{region '#Template'}
	{attribute 'Version' := '1.2.0.0'}
	{attribute 'Tags' := '"LCID": "1031", "Text": "DUT, Operation mode, Universal, On, Off"'}
	{attribute 'Tags' := '"LCID": "1033", "Text": "DUT, Operation mode, Universal, On, Off"'}
	{attribute 'Description' := '"LCID": "1031", "Text": "Betriebsart Ein Aus"'}
	{attribute 'Description' := '"LCID": "1033", "Text": "Operating on off"'}
{endregion}

{attribute qualified_only}
TYPE E_BA_OnOff :
(
	eOff			:= 1,
	eOn				:= 2
	
) UDINT;
END_TYPE

(* stored: Version 1.1.0.1, ProductVersion 3.1.4024.9
   DUT E_BA_OnOff: Id {21be6654-409e-476d-af71-1a65ea62fb53} *)
